// TIA Portal V16 export
// export: Created 2021-11-12T13:32:24.1677424Z, ExportSetting WithDefaults, DisplayName Totally Integrated Automation Portal, DisplayVersion V16 Update 3, DisplayName TIA Portal Version Control Interface, DisplayVersion V16 Update 2, DisplayName TIA Portal Openness, DisplayVersion V16 Update 3, DisplayName SINAMICS Startdrive Advanced, DisplayVersion V16 Update 5, DisplayName SINAMICS Startdrive G130, G150, S120, S150, SINAMICS MV, S210, DisplayVersion V16 Update 5, DisplayName SINAMICS Startdrive G110M, G120, G120C, G120D, G120P, G115D, DisplayVersion V16 Update 5, DisplayName STEP 7 Professional, DisplayVersion V16 Update 3, DisplayName STEP 7 Safety, DisplayVersion V16, DisplayName WinCC UA Professional, DisplayVersion V16 Update 3
DATA_BLOCK "HMI_CMD_KAS2"   // DB125
{ S7_Optimized_Access := 'TRUE' }
VERSION : 0.1
// stored: AutoNumber true, DBAccessibleFromOPCUA true, IsOnlyStoredInLoadMemory false, IsRetainMemResEnabled false, IsWriteProtectedInAS false, MemoryReserve 100
   VAR
      xxxxx__Others__xxxxx : Byte;
      NoOfPartsOk { S7_SetPoint := 'True'} : "UDT_PartCounter_Command";   // Number of OK parts
      NoOfPartsNotOk : "UDT_PartCounter_Command";   // Number of NOK parts
      EnableCutting : Bool;   // Manual enable in auto mode from HMI
      EnableLoading : Bool;   // Manual enable in auto mode from HMI
      xxxxx___SensorAlarms___xxxxx : Byte;
      LifeBit : "UDT_DI_Mon_Command";   // communication
      Saw { S7_SetPoint := 'True'} : "UDT_DI_Mon_Command";   // from saw
      ES { S7_SetPoint := 'True'} : "UDT_DI_Mon_Command";   // E-stop
   END_VAR
BEGIN
END_DATA_BLOCK
